// TIA Portal V20 export
DATA_BLOCK "T1-A ARUNC AUX"   // DB1902
{ S7_Optimized_Access := 'TRUE' }
// stored: AutoNumber false, MemoryReserve 100
   VAR
      AUX : Struct   // Auxiliary memory, not retentive memory
         "TIMER" : Array[1..50] of IEC_TIMER;
         OS : Array[0..50] of Bool;
         FO1 { S7_SetPoint := 'True'} : "FirstOut_aux";
      END_STRUCT;
   END_VAR
   VAR RETAIN
      AUX_MEMORY : Struct   // Auxiliary memory, retentive memory
         "BOOL" : Array[0..50] of Bool;
         "INT" : Array[0..20] of Int;
         "DINT" : Array[0..20] of DInt;
         "REAL" : Array[0..20] of Real;
      END_STRUCT;
   END_VAR
BEGIN
   // AUX."TIMER"[1] : Timer to delay the signal of the change diameter preset by LV2
END_DATA_BLOCK
